TYPE ST_History_HMI :
STRUCT
	iOK	:UDINT;
	iNOK :UDINT;
	bShift1	:BOOL;
	bShift2 :BOOL;
	bShift3 :BOOL;
END_STRUCT
END_TYPE

(* stored: Version 1.1.0.1
   DUT ST_History_HMI: Id {872ccca9-bede-4dc6-b7db-566268de70fe} *)
